FUNCTION_BLOCK EA_network2
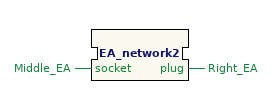
  SOCKETS
    socket : Middle_EA;
  END_SOCKETS
  PLUGS
    plug : Right_EA;
  END_PLUGS
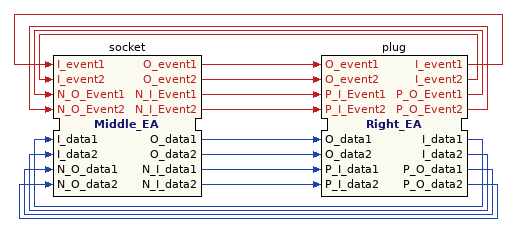
  EVENT_CONNECTIONS
    socket.O_event1 TO plug.O_event1;
    socket.O_event2 TO plug.O_event2;
    socket.N_I_Event1 TO plug.P_I_Event1;
    socket.N_I_Event2 TO plug.P_I_Event2;
    plug.I_event1 TO socket.I_event1;
    plug.I_event2 TO socket.I_event2;
    plug.P_O_Event1 TO socket.N_O_Event1;
    plug.P_O_Event2 TO socket.N_O_Event2;
  END_CONNECTIONS
  DATA_CONNECTIONS
    socket.O_data1 TO plug.O_data1;
    socket.O_data2 TO plug.O_data2;
    socket.N_I_data1 TO plug.P_I_data1;
    socket.N_I_data2 TO plug.P_I_data2;
    plug.I_data1 TO socket.I_data1;
    plug.I_data2 TO socket.I_data2;
    plug.P_O_data1 TO socket.N_O_data1;
    plug.P_O_data2 TO socket.N_O_data2;
  END_CONNECTIONS
END_FUNCTION_BLOCK
